FUNCTION_BLOCK Safe
VAR_INPUT
END_VAR
VAR_OUTPUT
END_VAR
VAR
END_VAR

// NETWORK 1

END_FUNCTION_BLOCK

(* stored: Version 1.1.0.1, ProductVersion 3.1.4024.11
   POU Safe: Id {ef7b8359-d872-4d31-807c-58a034359241}, SpecialFunc None *)
